// Mitsubishi GX Works2 project: projectPLC_NEW (2) (1)   PLC: FX3G

// global labels: Global1
VAR_GLOBAL
  X_System_Start AT X007 : BOOL;
  Y_System_On AT Y007 : BOOL;
  D_Cream_Start AT D1100 : INT;
  D_Chocolate_Start AT D1102 : INT;
  D_Biscuit_Start AT D1104 : INT;
  D_Cream_Container AT D1106 : INT;
  D_Cream_Machine AT D1108 : INT;
  D_Chocolate_Container AT D1110 : INT;
  D_Chocolate_Machine AT D1112 : INT;
  D_Biscuit_Container AT D1114 : INT;
  M_Initiate_Success AT M0 : BOOL;
  M_Cream_Success AT M1 : BOOL;
  M_Chocolate_Success AT M2 : BOOL;
  M_Biscuit_Success AT M3 : BOOL;
END_VAR
VAR_GLOBAL CONSTANT
  Const_Min_Cream : INT := 300;
  Const_Min_Chocolate : INT := 240;
  Const_Min_Biscuits : INT := 6;
END_VAR
VAR_GLOBAL
  X_MoveTo_Cream_Machine AT X011 : BOOL;
  M_Move_Cream_Success AT M11 : BOOL;
  M_Success_X11 AT M5 : BOOL;
END_VAR
VAR_GLOBAL CONSTANT
  Const_0 : INT;
END_VAR
VAR_GLOBAL
  M_Suc_move_biscuit AT M6 : BOOL;
  M_System_A_On AT M10 : BOOL;
  Sen_location AT X004 : BOOL;
  Sen_15 AT X002 : BOOL;
  Sen_30 AT X001 : BOOL;
  Y_Ziluf_On AT Y004 : BOOL;
  X_System_A_Start AT X010 : BOOL;
  M_30 AT M30 : BOOL;
  M_4 AT M4 : BOOL;
  D_Finish_Cream AT D1116 : INT;
  M_Finish_A AT M7 : BOOL;
END_VAR
VAR_GLOBAL CONSTANT
  Const_Timer_4s : INT := 40;
END_VAR
VAR_GLOBAL
  T_Timer_4s AT TC1 : BOOL;
  Ts_1 AT TS1 : BOOL;
  M_4sec_Finish AT M8 : BOOL;
  T_LightOne AT TC2 : BOOL;
  Ts_2 AT TS2 : BOOL;
  T_LightTwo AT TC3 : BOOL;
  Ts_3 AT TS3 : BOOL;
END_VAR
VAR_GLOBAL CONSTANT
  Const_Timer_1s : INT := 10;
END_VAR
VAR_GLOBAL
  Y_LightOne AT Y000 : BOOL;
  Y_LightTwo AT Y001 : BOOL;
  X_Stop_Ziluf AT X005 : BOOL;
  Sens_Camera AT X003 : BOOL;
  X_Start_B_Chocolate AT X006 : BOOL;
  M_9 AT M9 : BOOL;
  D_REAL_AnalogInput AT D8280 : INT;
  D_Saved_AnalogInput AT D8201 : INT;
END_VAR
VAR_GLOBAL CONSTANT
  Const_5 : INT := 5;
  Const_6 : INT := 6;
  Const_10 : INT := 10;
  Const_Reg_Choc : INT := 120;
END_VAR
VAR_GLOBAL
  M_Success_Chocolate_Dip1 AT M13 : BOOL;
  D_DIV_AnalogInput AT D8203 : INT;
  M_15 AT M15 : BOOL;
  M_Success_Chocolate_Dip2 AT M14 : BOOL;
  T_4 AT TC4 : BOOL;
  Ts_4 AT TS4 : BOOL;
END_VAR
VAR_GLOBAL CONSTANT
  Const_50 : INT := 50;
END_VAR
VAR_GLOBAL
  Y_Machine_B AT Y003 : BOOL;
  X_Wrapping AT X000 : BOOL;
  CC_Wrapping AT CC1 : BOOL;
  CS_Wrapping AT CS1 : BOOL;
  Y_Wrapping_At_5 AT Y002 : BOOL;
  CC_Temp_6 AT CC2 : BOOL;
  CS_Temp_6 AT CS2 : BOOL;
  M_under5 AT M100 : BOOL;
  M_120 AT M101 : BOOL;
  M_move120 AT M102 : BOOL;
  M_UP5 AT M103 : BOOL;
  M_240 AT M104 : BOOL;
  M_Move240 AT M105 : BOOL;
  M_finishB AT M106 : BOOL;
  M_EndOfDay AT M200 : BOOL;
  T_Timer_3sec AT TC5 : BOOL;
  Ts_5 AT TS5 : BOOL;
  T_Timer2_1sec AT TC6 : BOOL;
  Ts_6 AT TS6 : BOOL;
END_VAR
VAR_GLOBAL CONSTANT
  Const_3sec : INT := 30;
END_VAR
VAR_GLOBAL
  M_301 AT M301 : BOOL;
  M_ForY7 AT M302 : BOOL;
  M_add6_tocrembonum AT M304 : BOOL;
  D_output AT D8282 : INT;
  M_StartBlinkY7 AT M12 : BOOL;
  M_startSystem AT M17 : BOOL;
  M_blinking2 AT M303 : BOOL;
  T_timerTwo AT TC7 : BOOL;
  Ts_7 AT TS7 : BOOL;
  D_Krembo_Num AT D1198 : INT;
  M_Finish_analog AT M65 : BOOL;
  M_Reset11 AT M66 : BOOL;
  M_Y7 AT M55 : BOOL;
END_VAR
VAR_GLOBAL CONSTANT
  Constt_404 : INT := 404;
END_VAR
VAR_GLOBAL
  M_Help11 AT M78 : BOOL;
  M_Wrapping6 AT M79 : BOOL;
END_VAR

// task Task_01 (event TRUE, interval 0, priority 31): POU_01

PROGRAM POU_01
(* structured ladder/FBD written out as ST: instructions are called as NAME(EN, inputs, outputs); _pN, _eN, _tN stand for wires *)
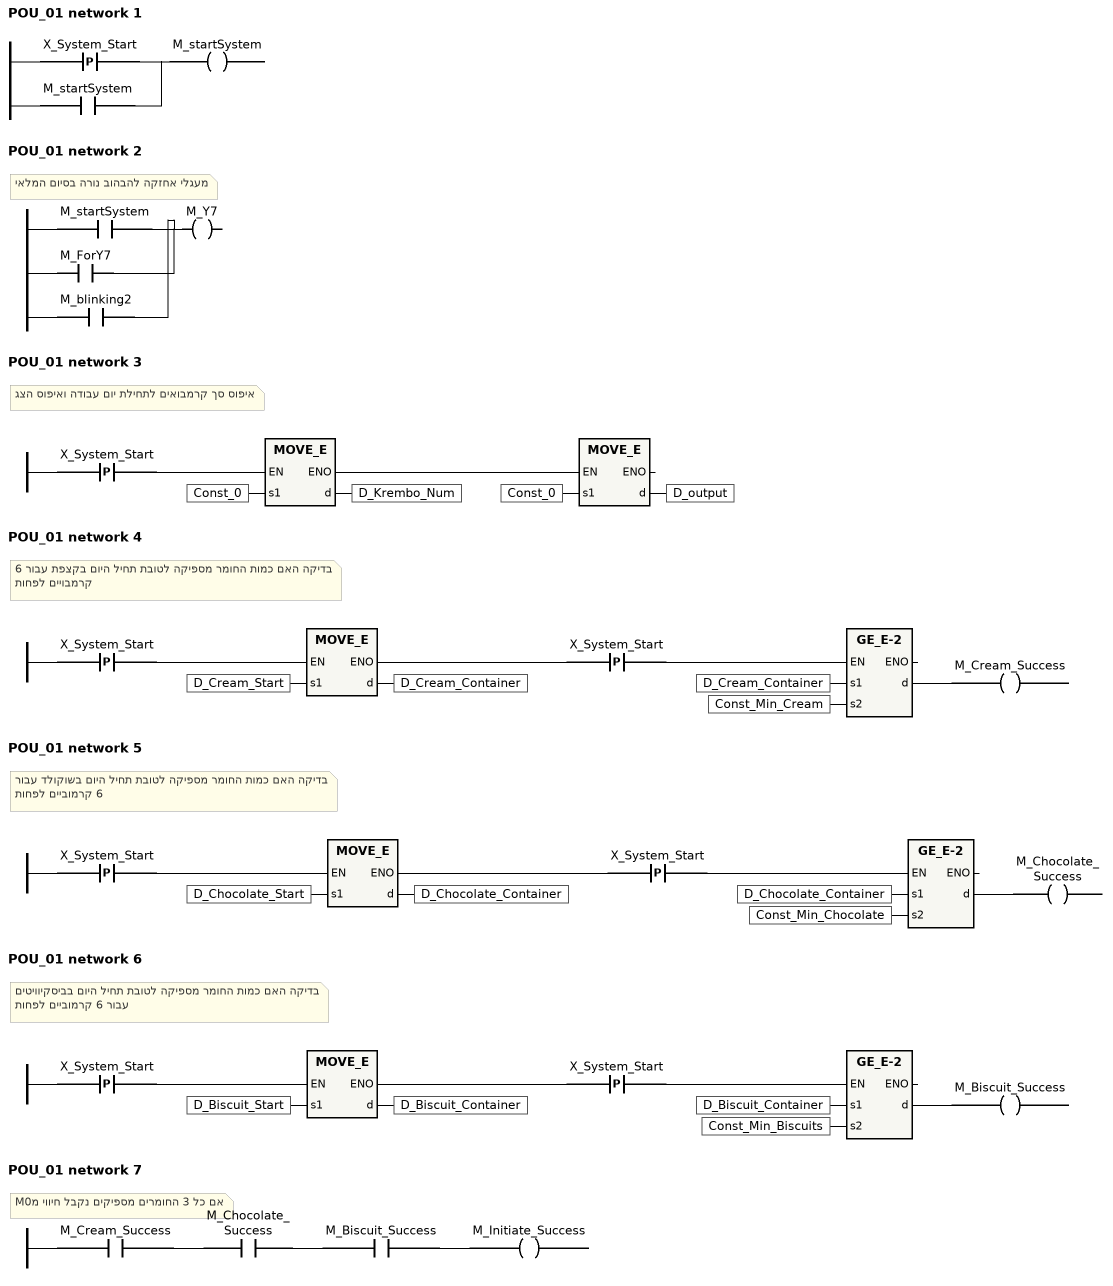
(* network 1 *)
M_startSystem := LDP(TRUE, X_System_Start) OR M_startSystem;
(* network 2 *)
(* מעגלי אחזקה להבהוב נורה בסיום המלאי *)
M_Y7 := M_startSystem OR M_ForY7 OR M_blinking2;
(* network 3 *)
(* איפוס סך קרמבואים לתחילת יום עבודה ואיפוס הצג *)
_e1 := MOVE_E(LDP(TRUE, X_System_Start), Const_0, D_Krembo_Num);
MOVE_E(_e1, Const_0, D_output);
(* network 4 *)
(* בדיקה האם כמות החומר מספיקה לטובת תחיל היום בקצפת עבור 6 קרמבויים לפחות *)
_e1 := MOVE_E(LDP(TRUE, X_System_Start), D_Cream_Start, D_Cream_Container);
GE_E(_e1 AND LDP(TRUE, X_System_Start), D_Cream_Container, Const_Min_Cream, _t2);
M_Cream_Success := _t2;
(* network 5 *)
(* בדיקה האם כמות החומר מספיקה לטובת תחיל היום בשוקולד עבור 6 קרמוביים לפחות *)
_e1 := MOVE_E(LDP(TRUE, X_System_Start), D_Chocolate_Start, D_Chocolate_Container);
GE_E(_e1 AND LDP(TRUE, X_System_Start), D_Chocolate_Container, Const_Min_Chocolate, _t2);
M_Chocolate_Success := _t2;
(* network 6 *)
(* בדיקה האם כמות החומר מספיקה לטובת תחיל היום בביסקיוויטים עבור 6 קרמוביים לפחות *)
_e1 := MOVE_E(LDP(TRUE, X_System_Start), D_Biscuit_Start, D_Biscuit_Container);
GE_E(_e1 AND LDP(TRUE, X_System_Start), D_Biscuit_Container, Const_Min_Biscuits, _t2);
M_Biscuit_Success := _t2;
(* network 7 *)
(* אם כל 3 החומרים מספיקים נקבל חיווי מM0 *)
M_Initiate_Success := M_Cream_Success AND M_Chocolate_Success AND M_Biscuit_Success;
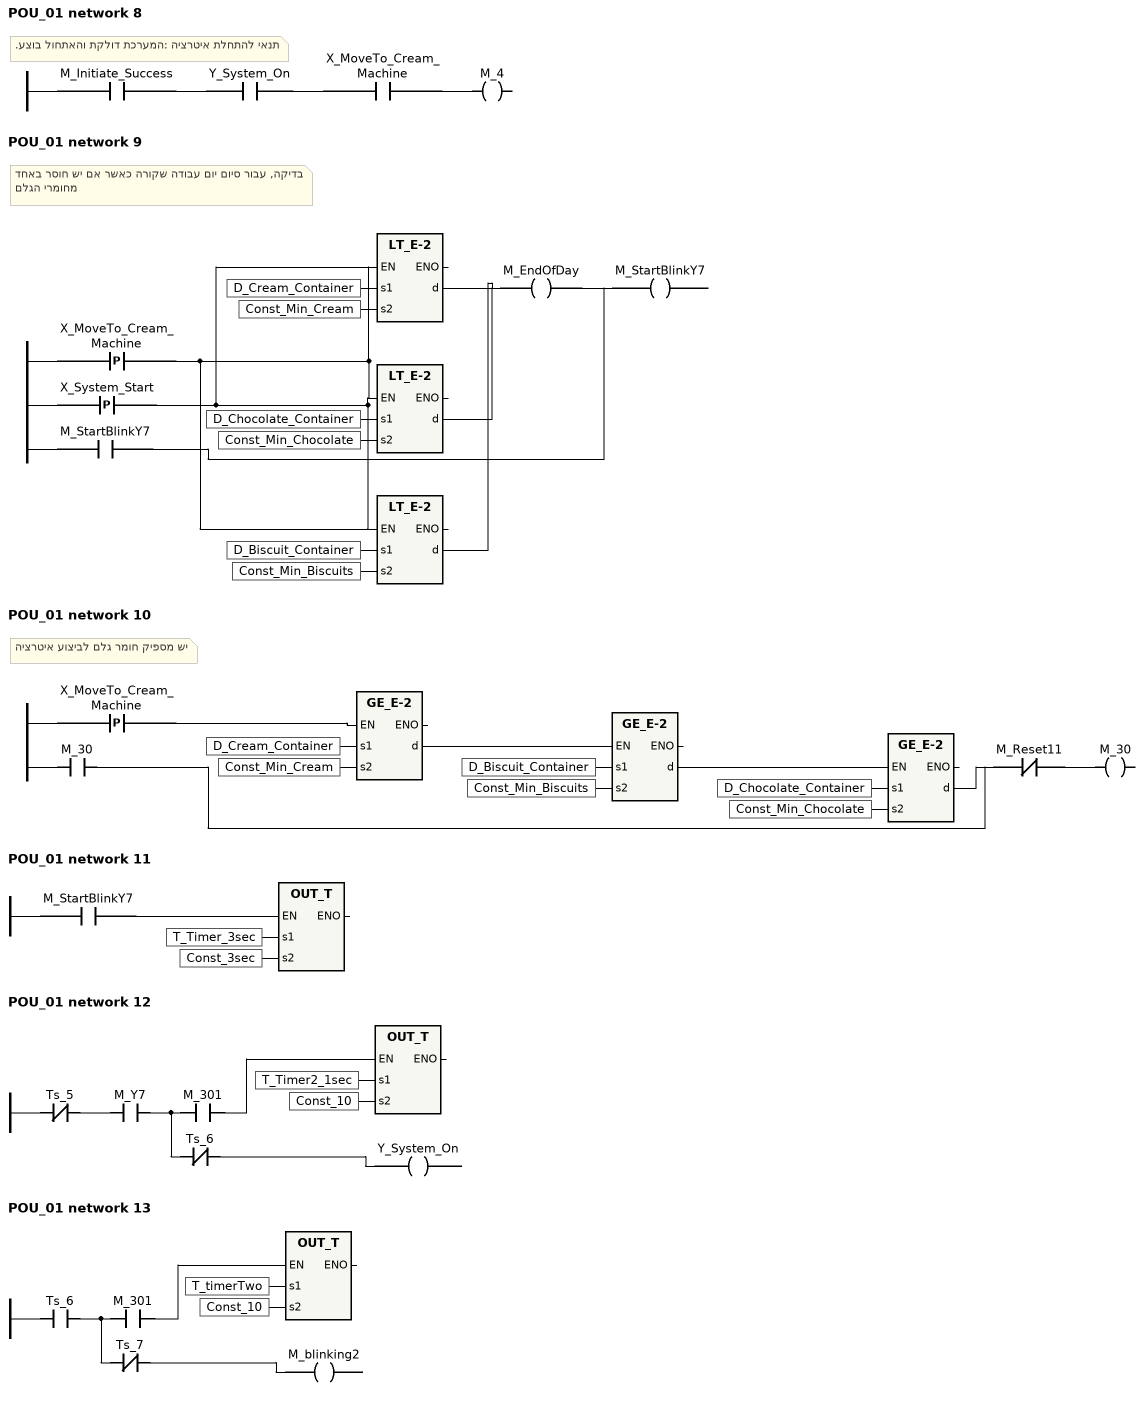
(* network 8 *)
(* תנאי להתחלת איטרציה :המערכת דולקת והאתחול בוצע. *)
M_4 := M_Initiate_Success AND Y_System_On AND X_MoveTo_Cream_Machine;
(* network 9 *)
(* בדיקה, עבור סיום יום עבודה שקורה כאשר אם יש חוסר באחד מחומרי הגלם *)
_p1 := LDP(TRUE, X_MoveTo_Cream_Machine) OR LDP(TRUE, X_System_Start);
LT_E(_p1, D_Cream_Container, Const_Min_Cream, _t2);
LT_E(_p1, D_Chocolate_Container, Const_Min_Chocolate, _t3);
LT_E(_p1, D_Biscuit_Container, Const_Min_Biscuits, _t4);
_p5 := _t2 OR _t3 OR _t4;
M_EndOfDay := _p5;
M_StartBlinkY7 := _p5 OR M_StartBlinkY7;
(* network 10 *)
(* יש מספיק חומר גלם לביצוע איטרציה *)
GE_E(LDP(TRUE, X_MoveTo_Cream_Machine), D_Cream_Container, Const_Min_Cream, _t1);
GE_E(_t1, D_Biscuit_Container, Const_Min_Biscuits, _t2);
GE_E(_t2, D_Chocolate_Container, Const_Min_Chocolate, _t3);
M_30 := (_t3 OR M_30) AND NOT M_Reset11;
(* network 11 *)
OUT_T(M_StartBlinkY7, T_Timer_3sec, Const_3sec);
(* network 12 *)
_p1 := NOT Ts_5 AND M_Y7;
OUT_T(_p1 AND M_301, T_Timer2_1sec, Const_10);
Y_System_On := _p1 AND NOT Ts_6;
(* network 13 *)
OUT_T(Ts_6 AND M_301, T_timerTwo, Const_10);
M_blinking2 := Ts_6 AND NOT Ts_7;
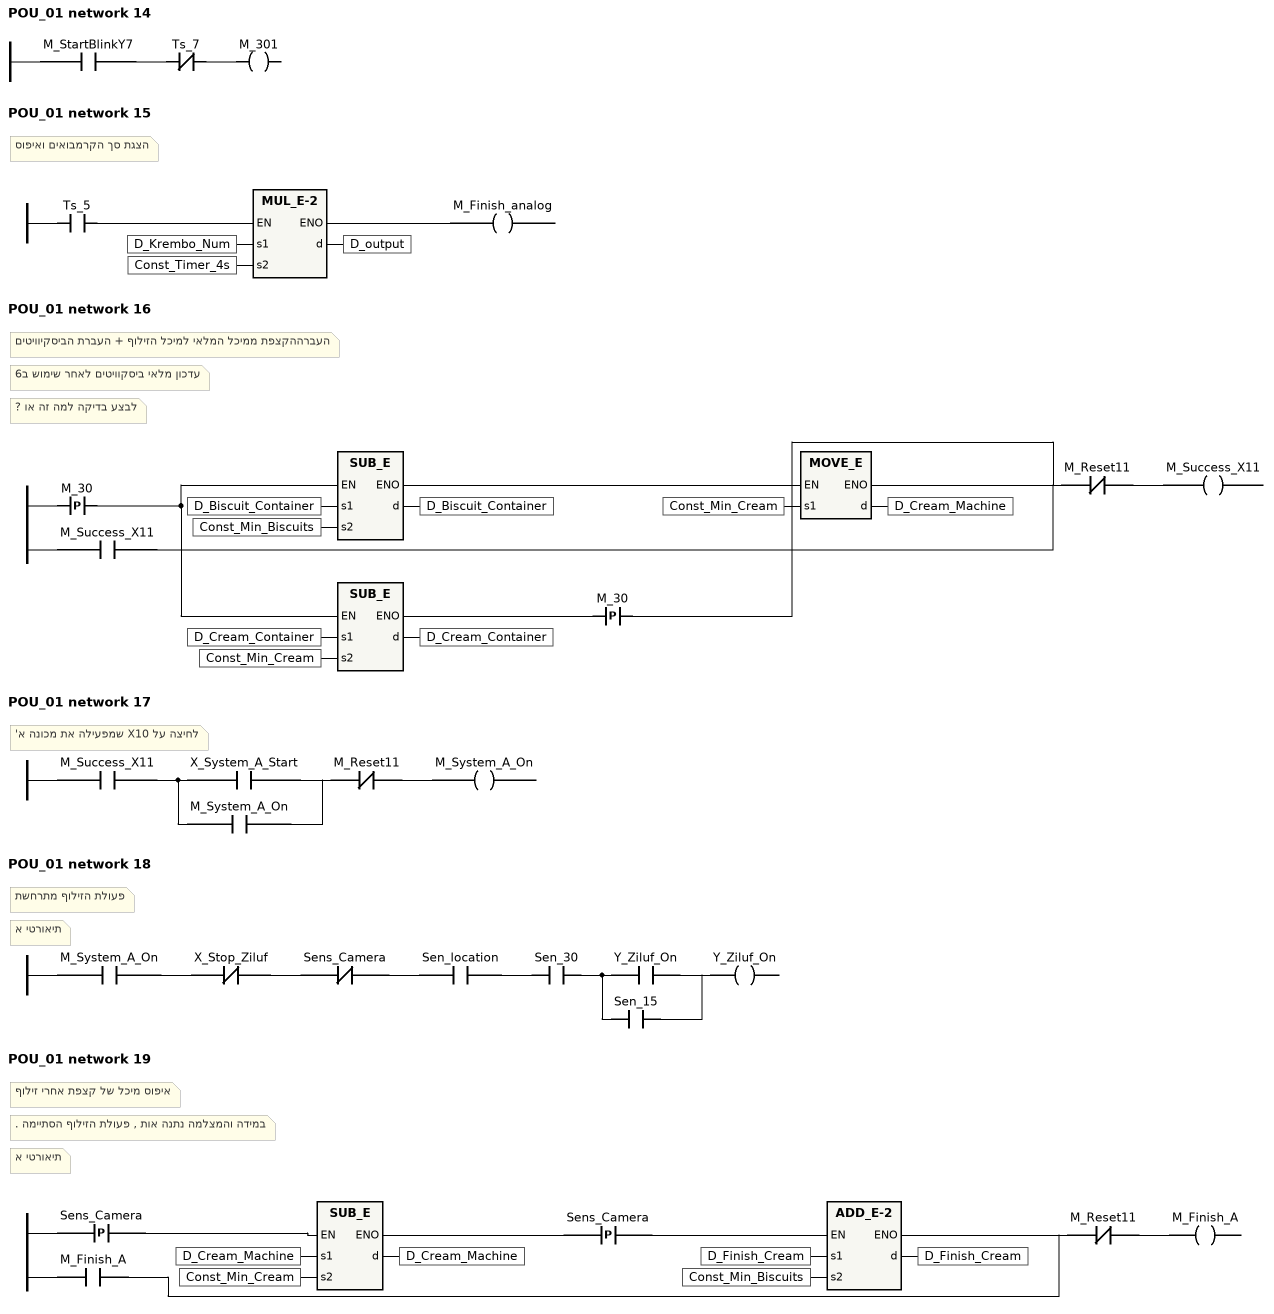
(* network 14 *)
M_301 := M_StartBlinkY7 AND NOT Ts_7;
(* network 15 *)
(* הצגת סך הקרמבואים ואיפוס *)
_e1 := MUL_E(Ts_5, D_Krembo_Num, Const_Timer_4s, D_output);
M_Finish_analog := _e1;
(* network 16 *)
(* העברההקצפת ממיכל המלאי למיכל הזילוף + העברת הביסקיוויטים *)
(* עדכון מלאי ביסקוויטים לאחר שימוש ב6 *)
(* לבצע בדיקה למה זה או ? *)
_p1 := LDP(TRUE, M_30);
_e2 := SUB_E(_p1, D_Cream_Container, Const_Min_Cream, D_Cream_Container);
_e3 := MOVE_E(_e2 AND LDP(TRUE, M_30), Const_Min_Cream, D_Cream_Machine);
_e4 := SUB_E(_p1, D_Biscuit_Container, Const_Min_Biscuits, D_Biscuit_Container);
M_Success_X11 := (_e3 OR _e4 OR M_Success_X11) AND NOT M_Reset11;
(* network 17 *)
(* לחיצה על X10 שמפעילה את מכונה א' *)
M_System_A_On := ((M_Success_X11 AND X_System_A_Start) OR (M_Success_X11 AND M_System_A_On)) AND NOT M_Reset11;
(* network 18 *)
(* פעולת הזילוף מתרחשת *)
(* תיאורטי א *)
_p1 := M_System_A_On AND NOT X_Stop_Ziluf AND NOT Sens_Camera AND Sen_location AND Sen_30;
Y_Ziluf_On := (_p1 AND Y_Ziluf_On) OR (_p1 AND Sen_15);
(* network 19 *)
(* איפוס מיכל של קצפת אחרי זילוף *)
(* במידה והמצלמה נתנה אות , פעולת הזילוף הסתיימה . *)
(* תיאורטי א *)
_e1 := SUB_E(LDP(TRUE, Sens_Camera), D_Cream_Machine, Const_Min_Cream, D_Cream_Machine);
_e2 := ADD_E(_e1 AND LDP(TRUE, Sens_Camera), D_Finish_Cream, Const_Min_Biscuits, D_Finish_Cream);
M_Finish_A := (_e2 OR M_Finish_A) AND NOT M_Reset11;
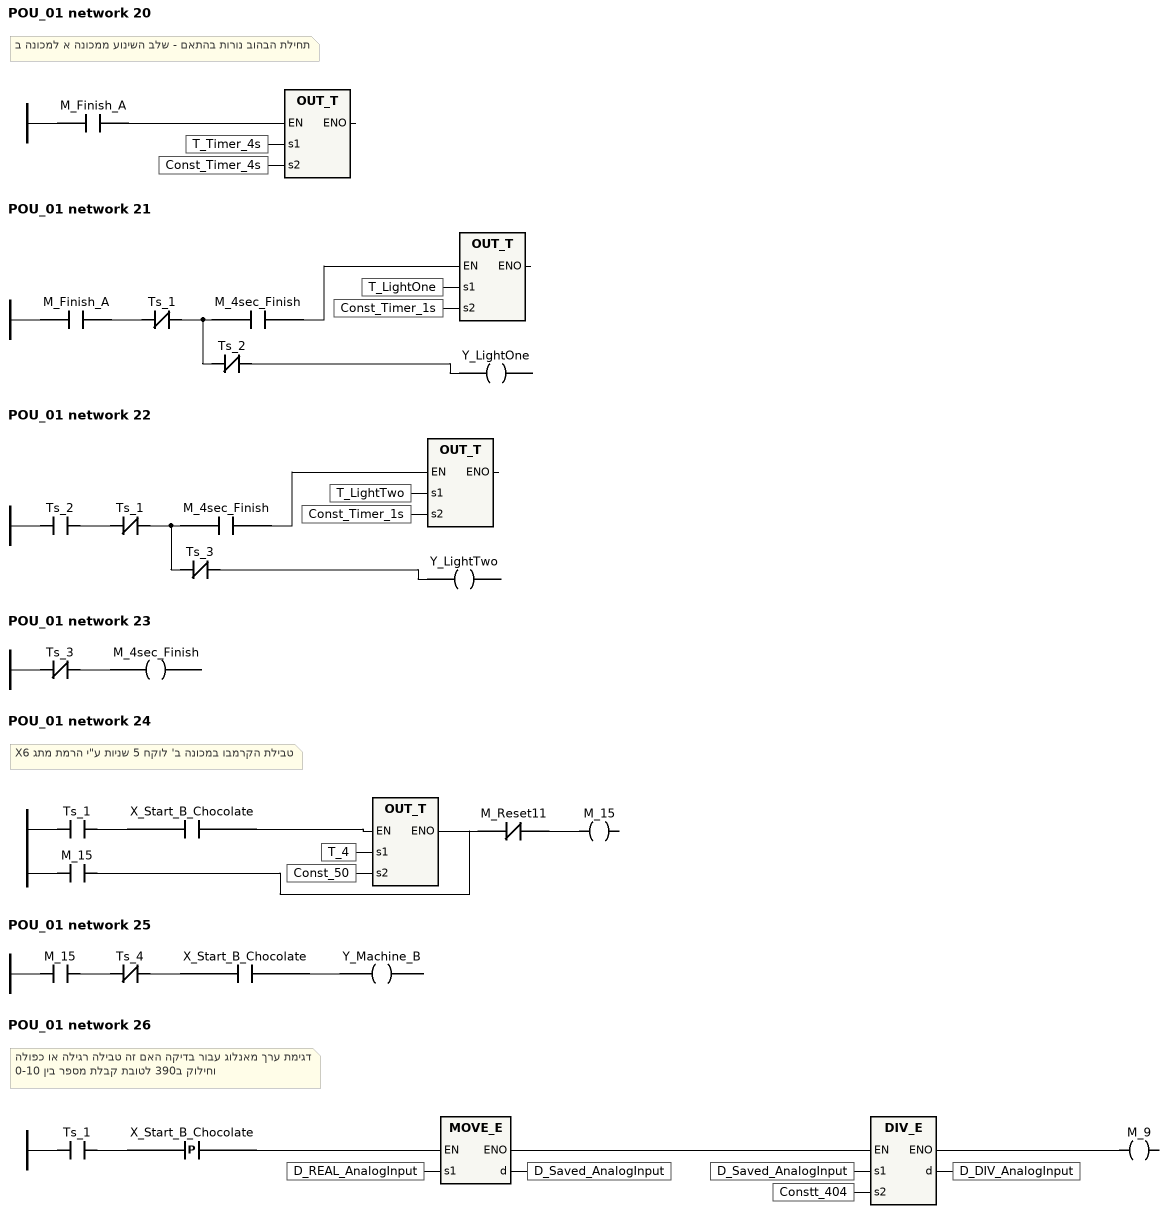
(* network 20 *)
(* תחילת הבהוב נורות בהתאם - שלב השינוע ממכונה א למכונה ב *)
OUT_T(M_Finish_A, T_Timer_4s, Const_Timer_4s);
(* network 21 *)
_p1 := M_Finish_A AND NOT Ts_1;
OUT_T(_p1 AND M_4sec_Finish, T_LightOne, Const_Timer_1s);
Y_LightOne := _p1 AND NOT Ts_2;
(* network 22 *)
_p1 := Ts_2 AND NOT Ts_1;
OUT_T(_p1 AND M_4sec_Finish, T_LightTwo, Const_Timer_1s);
Y_LightTwo := _p1 AND NOT Ts_3;
(* network 23 *)
M_4sec_Finish := NOT Ts_3;
(* network 24 *)
(* טבילת הקרמבו במכונה ב' לוקח 5 שניות ע"י הרמת מתג X6 *)
_e1 := OUT_T(Ts_1 AND X_Start_B_Chocolate, T_4, Const_50);
M_15 := (_e1 OR M_15) AND NOT M_Reset11;
(* network 25 *)
Y_Machine_B := M_15 AND NOT Ts_4 AND X_Start_B_Chocolate;
(* network 26 *)
(* דגימת ערך מאנלוג עבור בדיקה האם זה טבילה רגילה או כפולה וחילוק ב390 לטובת קבלת מספר בין 0-10 *)
_e1 := MOVE_E(Ts_1 AND LDP(TRUE, X_Start_B_Chocolate), D_REAL_AnalogInput, D_Saved_AnalogInput);
_e2 := DIV_E(_e1, D_Saved_AnalogInput, Constt_404, D_DIV_AnalogInput);
M_9 := _e2;
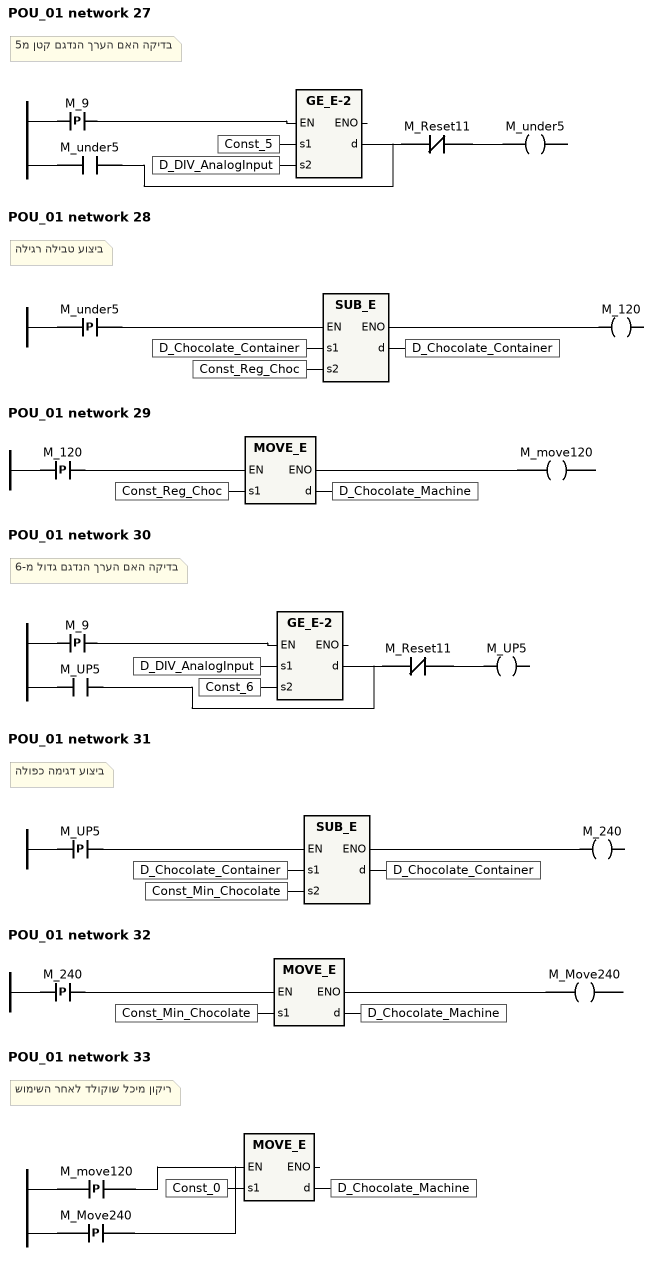
(* network 27 *)
(* בדיקה האם הערך הנדגם קטן מ5 *)
GE_E(LDP(TRUE, M_9), Const_5, D_DIV_AnalogInput, _t1);
M_under5 := (_t1 OR M_under5) AND NOT M_Reset11;
(* network 28 *)
(* ביצוע טבילה רגילה *)
_e1 := SUB_E(LDP(TRUE, M_under5), D_Chocolate_Container, Const_Reg_Choc, D_Chocolate_Container);
M_120 := _e1;
(* network 29 *)
_e1 := MOVE_E(LDP(TRUE, M_120), Const_Reg_Choc, D_Chocolate_Machine);
M_move120 := _e1;
(* network 30 *)
(* בדיקה האם הערך הנדגם גדול מ-6 *)
GE_E(LDP(TRUE, M_9), D_DIV_AnalogInput, Const_6, _t1);
M_UP5 := (_t1 OR M_UP5) AND NOT M_Reset11;
(* network 31 *)
(* ביצוע דגימה כפולה *)
_e1 := SUB_E(LDP(TRUE, M_UP5), D_Chocolate_Container, Const_Min_Chocolate, D_Chocolate_Container);
M_240 := _e1;
(* network 32 *)
_e1 := MOVE_E(LDP(TRUE, M_240), Const_Min_Chocolate, D_Chocolate_Machine);
M_Move240 := _e1;
(* network 33 *)
(* ריקון מיכל שוקולד לאחר השימוש *)
MOVE_E(LDP(TRUE, M_move120) OR LDP(TRUE, M_Move240), Const_0, D_Chocolate_Machine);
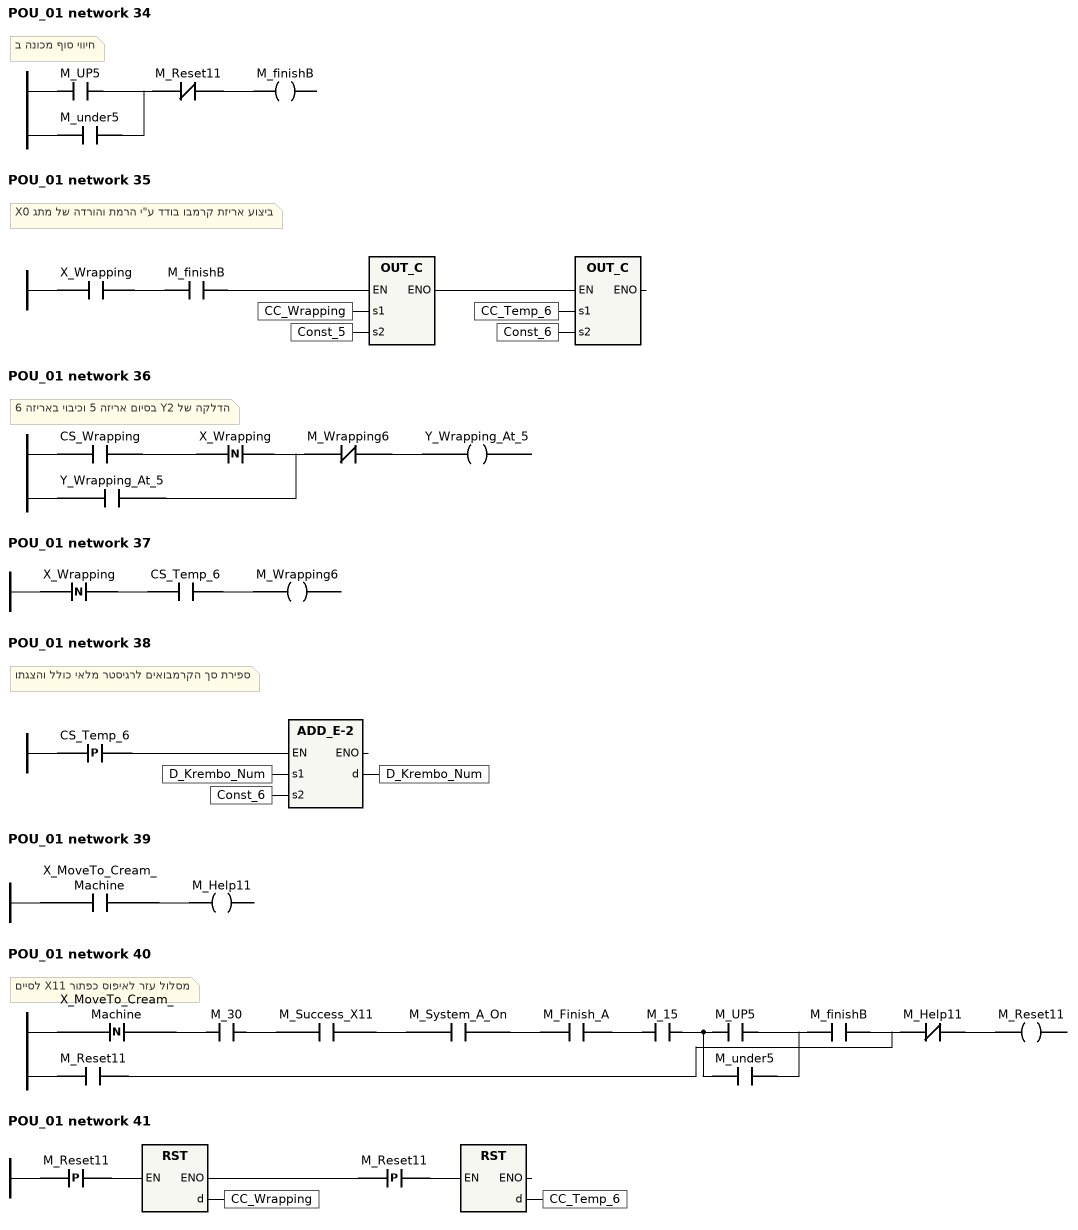
(* network 34 *)
(* חיווי סוף מכונה ב *)
M_finishB := (M_UP5 OR M_under5) AND NOT M_Reset11;
(* network 35 *)
(* ביצוע אריזת קרמבו בודד ע"י הרמת והורדה של מתג X0 *)
_e1 := OUT_C(X_Wrapping AND M_finishB, CC_Wrapping, Const_5);
OUT_C(_e1, CC_Temp_6, Const_6);
(* network 36 *)
(* הדלקה של Y2 בסיום אריזה 5 וכיבוי באריזה 6 *)
Y_Wrapping_At_5 := ((CS_Wrapping AND LDF(TRUE, X_Wrapping)) OR Y_Wrapping_At_5) AND NOT M_Wrapping6;
(* network 37 *)
M_Wrapping6 := LDF(TRUE, X_Wrapping) AND CS_Temp_6;
(* network 38 *)
(* ספירת סך הקרמבואים לרגיסטר מלאי כולל והצגתו *)
ADD_E(LDP(TRUE, CS_Temp_6), D_Krembo_Num, Const_6, D_Krembo_Num);
(* network 39 *)
M_Help11 := X_MoveTo_Cream_Machine;
(* network 40 *)
(* מסלול עזר לאיפוס כפתור X11 לסיים *)
_p1 := LDF(TRUE, X_MoveTo_Cream_Machine) AND M_30 AND M_Success_X11 AND M_System_A_On AND M_Finish_A AND M_15;
M_Reset11 := ((((_p1 AND M_UP5) OR (_p1 AND M_under5)) AND M_finishB) OR M_Reset11) AND NOT M_Help11;
(* network 41 *)
_e1 := RST(LDP(TRUE, M_Reset11), CC_Wrapping);
RST(_e1 AND LDP(TRUE, M_Reset11), CC_Temp_6);
END_PROGRAM
